// TIA Portal V19 export
TYPE "PositioningMachine_DataPers"
// stored: Access Published
   STRUCT
      AxisEncoderSelection_OK : Bool;
      AxisParameters_OK : Bool;
      AxisReloadPostion_OK : Bool;
      ActualPosition : LReal;
   END_STRUCT;
END_TYPE
